FUNCTION_BLOCK TT_model (* Basic Function Block Type *)
  (* Standard: 61499-2 *)
  (* Version 0.3, 2009-09-15, JHC, Holobloc Inc, Changed transition priorities. *)
  (* Version 0.2, 2003-12-04, JHC, Rockwell Automation, Renamed for better indexing. *)
  (* Version 0.1, 2002-11-05, JHC, Rockwell Automation, Corrected missing ST element in Algorithm REQ. *)
  (* Version 0.0, 2000-05-30, JHC, Rockwell Automation *)
  (* Compiler header: package fb.rt.dasdA1.A2.TurnTable; *)
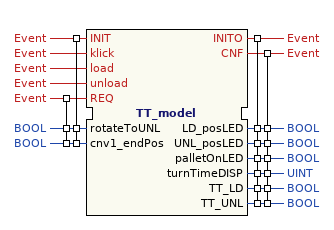
  EVENT_INPUT
    INIT WITH rotateToUNL, cnv1_endPos; (* Initialization Request *)
    klick;
    load;
    unload;
    REQ WITH rotateToUNL, cnv1_endPos;
  END_EVENT
  EVENT_OUTPUT
    INITO WITH LD_posLED, UNL_posLED, palletOnLED, turnTimeDISP, TT_LD, TT_UNL; (* Initialization Confirm *)
    CNF WITH LD_posLED, UNL_posLED, palletOnLED, turnTimeDISP, TT_LD, TT_UNL; (* Execution Confirmation *)
  END_EVENT
  VAR_INPUT
    rotateToUNL : BOOL;
    cnv1_endPos : BOOL;
  END_VAR
  VAR_OUTPUT
    LD_posLED : BOOL;
    UNL_posLED : BOOL;
    palletOnLED : BOOL;
    turnTimeDISP : UINT;
    TT_LD : BOOL;
    TT_UNL : BOOL;
  END_VAR
  VAR
    position : UINT := 1;
    palletON : BOOL := FALSE;
    turnOnProgress : BOOL := FALSE;
  END_VAR
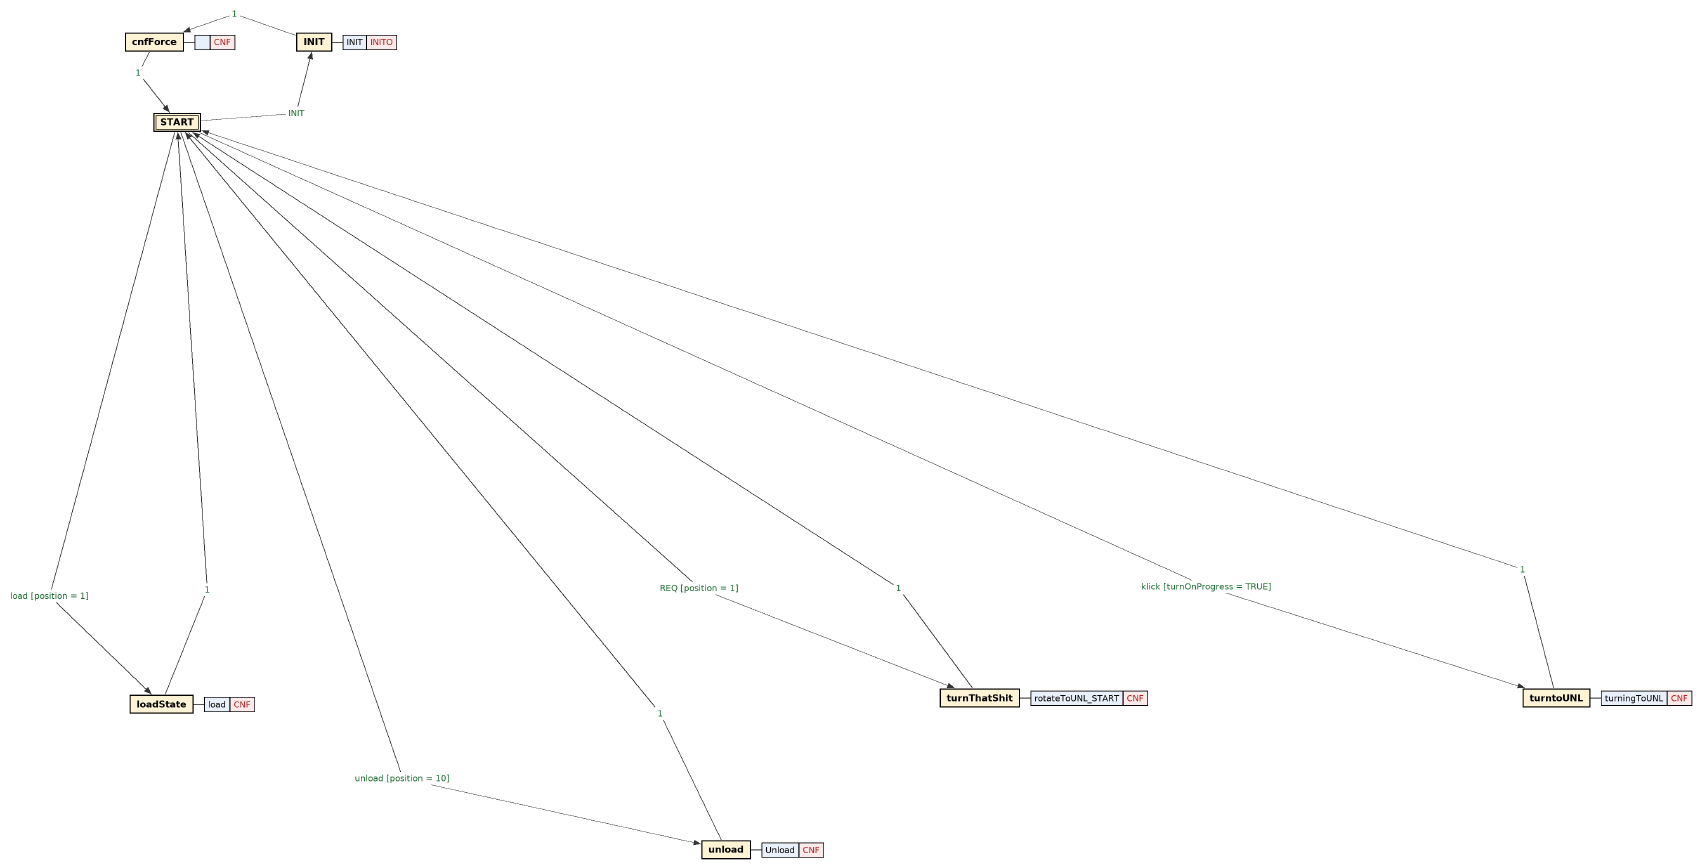
  EC_STATES
    START; (* Initial State *)
    INIT : INIT -> INITO; (* Initialization *)
    loadState : load -> CNF;
    unload : Unload -> CNF;
    turnThatShit : rotateToUNL_START -> CNF;
    turntoUNL : turningToUNL -> CNF;
    cnfForce : -> CNF;
  END_STATES
  EC_TRANSITIONS
    START TO INIT := INIT;
    START TO loadState := load [position = 1];
    loadState TO START := 1;
    START TO unload := unload [position = 10];
    unload TO START := 1;
    START TO turnThatShit := REQ [position = 1];
    turnThatShit TO START := 1;
    START TO turntoUNL := klick [turnOnProgress = TRUE];
    turntoUNL TO START := 1;
    INIT TO cnfForce := 1;
    cnfForce TO START := 1;
  END_TRANSITIONS
  ALGORITHM INIT IN ST: (* Initialization algorithm *)
LD_posLED := TRUE;
TT_LD := TRUE;
UNL_posLED := FALSE;
TT_UNL := FALSE;
palletON := FALSE;
  END_ALGORITHM
  ALGORITHM load IN ST:
IF (palletON = FALSE AND cnv1_endPos = TRUE) THEN
	palletON := TRUE;
	palletOnLED := TRUE;
END_IF;
  END_ALGORITHM
  ALGORITHM rotateToUNL_START IN ST:
turnOnProgress := TRUE;
  END_ALGORITHM
  ALGORITHM Unload IN ST:
IF (palletON = TRUE) THEN
	palletON := FALSE;
	palletOnLED := FALSE;
END_IF;
  END_ALGORITHM
  ALGORITHM turningToUNL IN ST:
IF (rotateToUNL = TRUE) THEN
	IF (position < 10) THEN
		TT_LD := FALSE;
		IF (position MOD 2 = 0) THEN
			UNL_posLED := TRUE;
			position := position + 1;
			turnTimeDISP := position;
		ELSE
			UNL_posLED := FALSE;
			position := position + 1;
			turnTimeDISP := position;
		END_IF;
	ELSE
		UNL_posLED := TRUE;
		TT_UNL := TRUE;
		LD_posLED := FALSE;
		TT_LD := FALSE;
	END_IF;
ELSE
	IF (position > 1) THEN
		TT_UNL := FALSE;
		IF (position MOD 2 = 0) THEN
			LD_posLED := TRUE;
			position := position - 1;
			turnTimeDISP := position;
		ELSE
			LD_posLED := FALSE;
			position := position - 1;
			turnTimeDISP := position;
		END_IF;
	ELSE
		UNL_posLED := FALSE;
		LD_posLED := TRUE;
		TT_LD := TRUE;
		turnOnProgress := FALSE;
	END_IF;

END_IF;
  END_ALGORITHM
END_FUNCTION_BLOCK
